{attribute 'qualified_only'}
{attribute 'strict'}
{attribute 'to_string'}
TYPE E_ClampingErrorCode :
(
    None                           := 16#0000,
    TorqueCommandRejected          := 16#7201,
    EnterTorqueModeTimeout         := 16#7202,
    AxisFaultDuringTorqueBuild     := 16#7203,
    TorqueBuildTimeout             := 16#7204,
    InvalidProcessStep             := 16#7205,
    PositionCommandNotReleased     := 16#7206,
    AxisFaultRestoringPosition     := 16#7207,
    RestorePositionModeTimeout     := 16#7208,
    HoldPositionCommandFailed      := 16#7209,
    PositionTimeout                := 16#720A // 夹紧轴松开、接近或保持定位超时
) UDINT;
END_TYPE

(* stored: Version 1.1.0.1, ProductVersion 3.1.4026.20
   DUT E_ClampingErrorCode: Id {d4d68bdf-eff9-46c5-926a-70d89951d815} *)
